// TIA Portal V17 export
// export: Created 2023-12-22T15:03:00.6243464Z, ExportSetting WithDefaults, DisplayName Totally Integrated Automation Portal, DisplayVersion V17, DisplayName TIA Portal Openness, DisplayVersion V17, DisplayName TIA Portal Version Control Interface, DisplayVersion V17, DisplayName STEP 7 Professional, DisplayVersion V17, DisplayName STEP 7 Safety, DisplayVersion V17, DisplayName WinCC Advanced, DisplayVersion V17
FUNCTION_BLOCK "DRV_M_D"   // FB110, LAD
{ S7_Optimized_Access := 'FALSE' }
VERSION : 0.1
// stored: AutoNumber false, IsIECCheckEnabled false, SetENOAutomatically false, UDAEnableTagReadback false
   VAR_INPUT
      All_Block : Bool;   // Аварийный останов
   END_VAR
   VAR_IN_OUT
      FB_QF : Bool;   // защитный автомат / Защитный автомат / Готовность
      FB_KM : Bool;   // привод запущен / Пускатель / В работе
      S_Alarm : Bool;   // Внешний индикатор наличия аварии
      CMD_Run : Bool;   // Команда запуска двигателя
   END_VAR
   VAR DB_SPECIFIC
      CMD : "CMD";   // Основные команды / Блок команд
      Mode : Int;   // Режим работы
      Status : Int;   // Статус устройства
      Use : Struct   // Функционал
         QF { S7_SetPoint := 'True'} : Bool := true;   // Защитный автомат
         KM { S7_SetPoint := 'True'} : Bool := true;   // Пускатель
         OpTime { S7_SetPoint := 'True'} : Bool := true;   // Контроль наработки
         Analog { S7_SetPoint := 'True'} : Bool;
         Local_Keys : Bool;
      END_STRUCT;
      FB : Struct   // Функционал
         QF : Bool;   // Защитный автомат
         KM : Bool;   // Пускатель
         Local_Start : Bool;
         Local_Stop : Bool;
      END_STRUCT;
      ON : Bool;   // Успешно запущено
      OFF : Bool;   // Успешно остановлено
   END_VAR
   VAR
      Tx { S7_SetPoint := 'True'} : Array[0..3] of "Time_S";   // Блок таймеров
   END_VAR
   VAR DB_SPECIFIC
      Inv : Struct   // Инверсия сигналов
         CMD { S7_SetPoint := 'True'} : Bool;   // Команда запуска
         QF { S7_SetPoint := 'True'} : Bool;   // Защитный автомат
         KM { S7_SetPoint := 'True'} : Bool;   // Пускатель
      END_STRUCT;
      Alarm : Struct   // Сбор аварий / Список аварий
         Block : Bool;   // Аварийная остановка
         QF : Bool;   // привод не готов / Выбило защитный автомат
         Start : Bool;   // Ошибка при запуске
         Stop : Bool;   // Ошибка при останове
         Termo : Bool;   // термозащита / Сработала термозащита
         Alarm : Bool;   // Внешняя авария
         Safety : Bool;   // Сработала безопасность
         OpTime : Bool;
      END_STRUCT;
      Alarms : Word;   // Слово аварий
      Events : Word;   // События
      pos : Array[0..15] of Bool;
      OpTime_h : DInt;   // наработка (ч)
      OpTime_s { S7_SetPoint := 'True'} : DInt;   // наработка (с)
      OpTime_SP { S7_SetPoint := 'True'} : DInt := 2160;   // Интервал обслуживания, ч
      OpTime_Now_h : DInt;   // Прошло с прошлого обслуживания, ч
      OpTime_Now_s { S7_SetPoint := 'True'} : DInt;   // Прошло с прошлого обслуживания, с
      CodeID { S7_SetPoint := 'True'} : Int;   // Код датчика для привязки в скаде
      Indirect : Struct   // Использование косвенной адресации
         FB_QF { S7_SetPoint := 'True'} : Bool := true;   // Защитный автомат
         FB_KM { S7_SetPoint := 'True'} : Bool := true;   // Пускатель
         CMD { S7_SetPoint := 'True'} : Bool := true;   // Запуск двигателя
      END_STRUCT;
      Indirect_BYTE : Struct   // Адрес входа на контроллере (Байт)
         FB_QF { S7_SetPoint := 'True'} : Int;   // Защитный автомат
         FB_KM { S7_SetPoint := 'True'} : Int;   // Пускатель
         CMD { S7_SetPoint := 'True'} : Int;   // Запуск двигателя
      END_STRUCT;
      Indirect_BIT : Struct   // Адрес входа на контроллере (Бит)
         FB_QF { S7_SetPoint := 'True'} : Int := 9;   // Защитный автомат
         FB_KM { S7_SetPoint := 'True'} : Int := 9;   // Пускатель
         CMD { S7_SetPoint := 'True'} : Int := 9;   // Запуск двигателя
      END_STRUCT;
      Time_DTL : DTL;
   END_VAR
   VAR_TEMP
      ev : Bool;
      xQF : Bool;
      xKM : Bool;
   END_VAR
   VAR_TEMP   // added for the SCL form of the ladder/FBD networks
      _w1 : Bool;
      _w2 : Bool;
      _w3 : Bool;
      _w4 : Bool;
      _w5 : Bool;
      _w6 : Bool;
      _w7 : Bool;
      _w8 : Bool;
      _w9 : Bool;
      _w10 : Bool;
      _w11 : Bool;
      _w12 : Bool;
      _w13 : Bool;
      _w14 : Bool;
      _w15 : Bool;
      _w16 : Bool;
      _w17 : Bool;
      _w18 : Bool;
      _w19 : Bool;
      _w20 : Bool;
      _w21 : Bool;
      _w22 : Bool;
      _w23 : Bool;
      _w24 : Bool;
      _w25 : Bool;
      _w26 : Bool;
   END_VAR
BEGIN

REGION Network 1: Режим глобальной симуляции
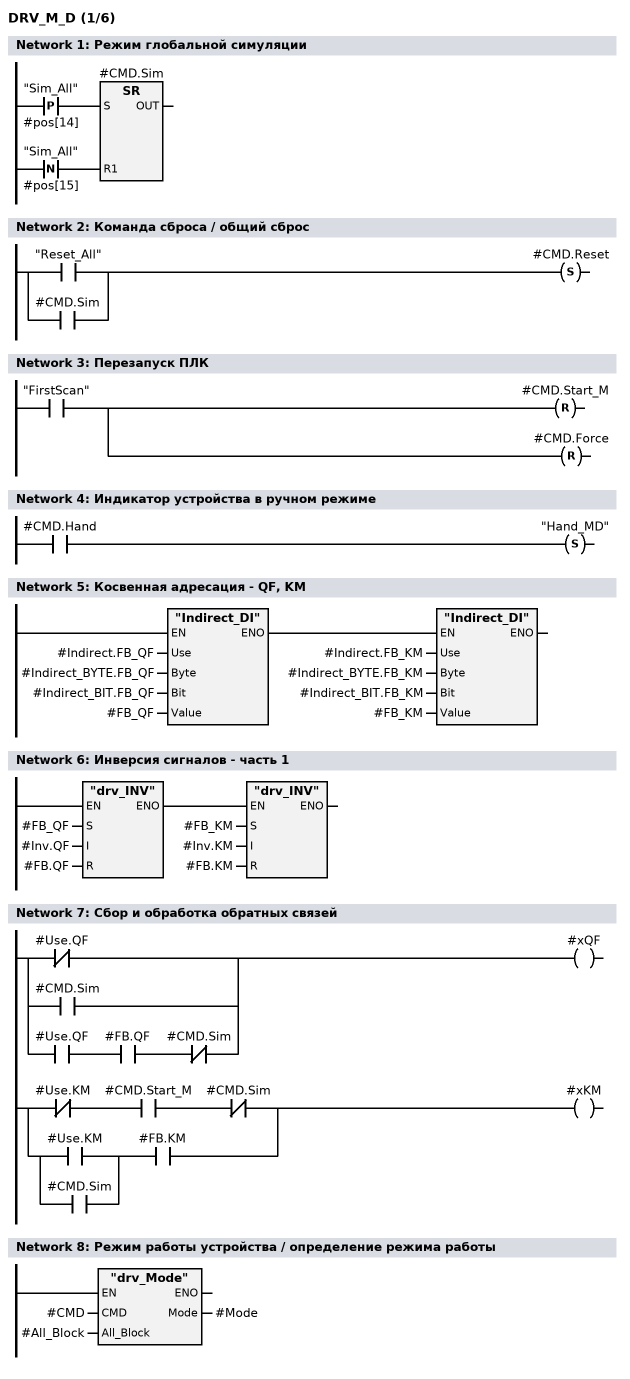
   RUNG wire#powerrail
      P_Contact(operand := "Sim_All", bit := #pos[14])
      S_SR(operand := #CMD.Sim, r1 := wire#w1)
   END_RUNG
   RUNG wire#powerrail
      N_Contact(operand := "Sim_All", bit := #pos[15])
   END_RUNG wire#w1
   // the same network as SCL:
   #_w1 := "Sim_All" AND NOT #pos[14];   // rising edge of "Sim_All"
   #pos[14] := "Sim_All";
   #_w2 := NOT "Sim_All" AND #pos[15];   // falling edge of "Sim_All"
   #pos[15] := "Sim_All";
   IF #_w1 THEN
       #CMD.Sim := TRUE;   // SR flip-flop
   END_IF;
   IF #_w2 THEN #CMD.Sim := FALSE; END_IF;
END_REGION

REGION Network 2: Команда сброса / общий сброс
   RUNG wire#powerrail
      Contact( "Reset_All" )
      wire#w1
      S_Coil( #CMD.Reset )
   END_RUNG
   RUNG wire#powerrail
      Contact( #CMD.Sim )
   END_RUNG wire#w1
   // the same network as SCL:
   IF "Reset_All" OR #CMD.Sim THEN #CMD.Reset := TRUE; END_IF;
END_REGION

REGION Network 3: Перезапуск ПЛК
   RUNG wire#powerrail
      Contact( "FirstScan" )
      wire#w1
      R_Coil( #CMD.Start_M )
   END_RUNG
   RUNG wire#w1
      R_Coil( #CMD.Force )
   END_RUNG
   // the same network as SCL:
   IF "FirstScan" THEN
       #CMD.Start_M := FALSE;
       #CMD.Force := FALSE;
   END_IF;
END_REGION

REGION Network 4: Индикатор устройства в ручном режиме
   RUNG wire#powerrail
      Contact( #CMD.Hand )
      S_Coil( "Hand_MD" )
   END_RUNG
   // the same network as SCL:
   IF #CMD.Hand THEN "Hand_MD" := TRUE; END_IF;
END_REGION

REGION Network 5: Косвенная адресация - QF, KM
   RUNG wire#powerrail
      "Indirect_DI"(Use := #Indirect.FB_QF, "Byte" := #Indirect_BYTE.FB_QF, Bit := #Indirect_BIT.FB_QF, Value := #FB_QF)
      "Indirect_DI"(Use := #Indirect.FB_KM, "Byte" := #Indirect_BYTE.FB_KM, Bit := #Indirect_BIT.FB_KM, Value := #FB_KM)
   END_RUNG
   // the same network as SCL:
   "Indirect_DI"(Use := #Indirect.FB_QF,
                 "Byte" := #Indirect_BYTE.FB_QF,
                 Bit := #Indirect_BIT.FB_QF,
                 Value := #FB_QF,
                 ENO => #_w1);
   IF #_w1 THEN
       "Indirect_DI"(Use := #Indirect.FB_KM,
                     "Byte" := #Indirect_BYTE.FB_KM,
                     Bit := #Indirect_BIT.FB_KM,
                     Value := #FB_KM);
   END_IF;
END_REGION

REGION Network 6: Инверсия сигналов - часть 1
   RUNG wire#powerrail
      "drv_INV"(S := #FB_QF, I := #Inv.QF, R := #FB.QF)
      "drv_INV"(S := #FB_KM, I := #Inv.KM, R := #FB.KM)
   END_RUNG
   // the same network as SCL:
   "drv_INV"(S := #FB_QF, I := #Inv.QF, R := #FB.QF, ENO => #_w1);
   IF #_w1 THEN "drv_INV"(S := #FB_KM, I := #Inv.KM, R := #FB.KM); END_IF;
END_REGION

REGION Network 7: Сбор и обработка обратных связей
   RUNG wire#powerrail
      I_Contact( #Use.QF )
      wire#w1
      Coil( #xQF )
   END_RUNG
   RUNG wire#powerrail
      Contact( #CMD.Sim )
   END_RUNG wire#w1
   RUNG wire#powerrail
      Contact( #Use.QF )
      Contact( #FB.QF )
      I_Contact( #CMD.Sim )
   END_RUNG wire#w1
   RUNG wire#powerrail
      I_Contact( #Use.KM )
      Contact( #CMD.Start_M )
      I_Contact( #CMD.Sim )
      wire#w2
      Coil( #xKM )
   END_RUNG
   RUNG wire#powerrail
      Contact( #Use.KM )
      wire#w3
      Contact( #FB.KM )
   END_RUNG wire#w2
   RUNG wire#powerrail
      Contact( #CMD.Sim )
   END_RUNG wire#w3
   // the same network as SCL:
   #xQF := NOT #Use.QF OR #CMD.Sim OR (#Use.QF AND #FB.QF AND NOT #CMD.Sim);
   #xKM := (NOT #Use.KM AND #CMD.Start_M AND NOT #CMD.Sim) OR ((#Use.KM OR #CMD.Sim) AND #FB.KM);
END_REGION

REGION Network 8: Режим работы устройства / определение режима работы
   RUNG wire#powerrail
      "drv_Mode"(CMD := #CMD, All_Block := #All_Block, Mode => #Mode)
   END_RUNG
   // the same network as SCL:
   "drv_Mode"(CMD := #CMD, All_Block := #All_Block, Mode => #Mode);
END_REGION

REGION Network 9: Управление запуском / дискретный управляющий сигнал
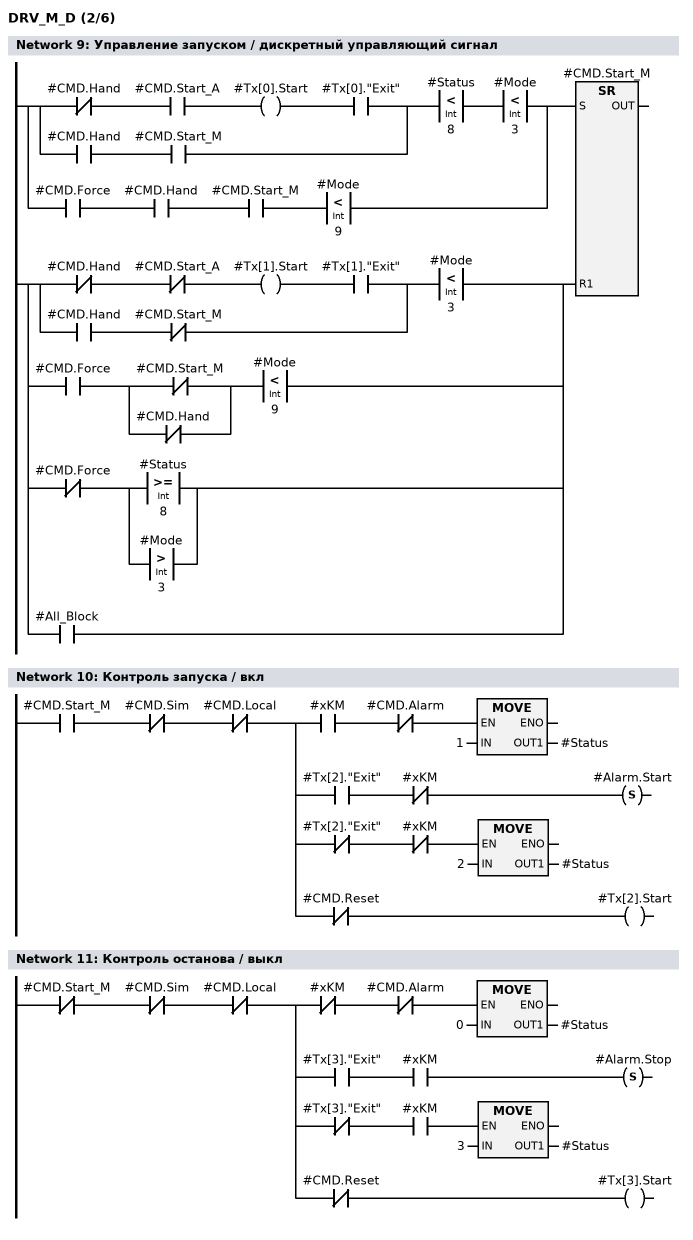
   RUNG wire#powerrail
      I_Contact( #CMD.Hand )
      Contact( #CMD.Start_A )
      Coil( #Tx[0].Start )
      Contact( #Tx[0]."Exit" )
      wire#w1
      { S7_Templates := "SrcType := Int" } LT_Contact(in1 := #Status, in2 := 8)
      { S7_Templates := "SrcType := Int" } LT_Contact(in1 := #Mode, in2 := 3)
      wire#w2
      S_SR(operand := #CMD.Start_M, r1 := wire#w7)
   END_RUNG
   RUNG wire#powerrail
      Contact( #CMD.Hand )
      Contact( #CMD.Start_M )
   END_RUNG wire#w1
   RUNG wire#powerrail
      Contact( #CMD.Force )
      Contact( #CMD.Hand )
      Contact( #CMD.Start_M )
      { S7_Templates := "SrcType := Int" } LT_Contact(in1 := #Mode, in2 := 9)
   END_RUNG wire#w2
   RUNG wire#powerrail
      I_Contact( #CMD.Hand )
      I_Contact( #CMD.Start_A )
      Coil( #Tx[1].Start )
      Contact( #Tx[1]."Exit" )
      wire#w3
      { S7_Templates := "SrcType := Int" } LT_Contact(in1 := #Mode, in2 := 3)
   END_RUNG wire#w7
   RUNG wire#powerrail
      Contact( #CMD.Hand )
      I_Contact( #CMD.Start_M )
   END_RUNG wire#w3
   RUNG wire#powerrail
      Contact( #CMD.Force )
      wire#w4
      I_Contact( #CMD.Start_M )
      wire#w5
      { S7_Templates := "SrcType := Int" } LT_Contact(in1 := #Mode, in2 := 9)
   END_RUNG wire#w7
   RUNG wire#w4
      I_Contact( #CMD.Hand )
   END_RUNG wire#w5
   RUNG wire#powerrail
      I_Contact( #CMD.Force )
      wire#w6
      { S7_Templates := "SrcType := Int" } GE_Contact(in1 := #Status, in2 := 8)
   END_RUNG wire#w7
   RUNG wire#w6
      { S7_Templates := "SrcType := Int" } GT_Contact(in1 := #Mode, in2 := 3)
   END_RUNG wire#w7
   RUNG wire#powerrail
      Contact( #All_Block )
   END_RUNG wire#w7
   // the same network as SCL:
   #Tx[0].Start := NOT #CMD.Hand AND #CMD.Start_A;
   #_w1 := (((NOT #CMD.Hand AND #CMD.Start_A AND #Tx[0]."Exit") OR (#CMD.Hand AND #CMD.Start_M)) AND (#Status < 8) AND (#Mode < 3)) OR (#CMD.Force AND #CMD.Hand AND #CMD.Start_M AND (#Mode < 9));
   #Tx[1].Start := NOT #CMD.Hand AND NOT #CMD.Start_A;
   #_w2 := (((NOT #CMD.Hand AND NOT #CMD.Start_A AND #Tx[1]."Exit") OR (#CMD.Hand AND NOT #CMD.Start_M)) AND (#Mode < 3)) OR (#CMD.Force AND (NOT #CMD.Start_M OR NOT #CMD.Hand) AND (#Mode < 9)) OR (NOT #CMD.Force AND ((#Status >= 8) OR (#Mode > 3))) OR #All_Block;
   IF #_w1 THEN
       #CMD.Start_M := TRUE;   // SR flip-flop
   END_IF;
   IF #_w2 THEN #CMD.Start_M := FALSE; END_IF;
END_REGION

REGION Network 10: Контроль запуска / вкл
   RUNG wire#powerrail
      Contact( #CMD.Start_M )
      I_Contact( #CMD.Sim )
      I_Contact( #CMD.Local )
      wire#w1
      Contact( #xKM )
      I_Contact( #CMD.Alarm )
      { S7_GenerateENO := "TRUE" } Move(in := 1, out1 => #Status)
   END_RUNG
   RUNG wire#w1
      Contact( #Tx[2]."Exit" )
      I_Contact( #xKM )
      S_Coil( #Alarm.Start )
   END_RUNG
   RUNG wire#w1
      I_Contact( #Tx[2]."Exit" )
      I_Contact( #xKM )
      { S7_GenerateENO := "TRUE" } Move(in := 2, out1 => #Status)
   END_RUNG
   RUNG wire#w1
      I_Contact( #CMD.Reset )
      Coil( #Tx[2].Start )
   END_RUNG
   // the same network as SCL:
   #_w1 := #CMD.Start_M AND NOT #CMD.Sim AND NOT #CMD.Local;
   IF #_w1 AND #xKM AND NOT #CMD.Alarm THEN #Status := 1; END_IF;
   IF #_w1 AND #Tx[2]."Exit" AND NOT #xKM THEN #Alarm.Start := TRUE; END_IF;
   IF #_w1 AND NOT #Tx[2]."Exit" AND NOT #xKM THEN #Status := 2; END_IF;
   #Tx[2].Start := #_w1 AND NOT #CMD.Reset;
END_REGION

REGION Network 11: Контроль останова / выкл
   RUNG wire#powerrail
      I_Contact( #CMD.Start_M )
      I_Contact( #CMD.Sim )
      I_Contact( #CMD.Local )
      wire#w1
      I_Contact( #xKM )
      I_Contact( #CMD.Alarm )
      { S7_GenerateENO := "TRUE" } Move(in := 0, out1 => #Status)
   END_RUNG
   RUNG wire#w1
      Contact( #Tx[3]."Exit" )
      Contact( #xKM )
      S_Coil( #Alarm.Stop )
   END_RUNG
   RUNG wire#w1
      I_Contact( #Tx[3]."Exit" )
      Contact( #xKM )
      { S7_GenerateENO := "TRUE" } Move(in := 3, out1 => #Status)
   END_RUNG
   RUNG wire#w1
      I_Contact( #CMD.Reset )
      Coil( #Tx[3].Start )
   END_RUNG
   // the same network as SCL:
   #_w1 := NOT #CMD.Start_M AND NOT #CMD.Sim AND NOT #CMD.Local;
   IF #_w1 AND NOT #xKM AND NOT #CMD.Alarm THEN #Status := 0; END_IF;
   IF #_w1 AND #Tx[3]."Exit" AND #xKM THEN #Alarm.Stop := TRUE; END_IF;
   IF #_w1 AND NOT #Tx[3]."Exit" AND #xKM THEN #Status := 3; END_IF;
   #Tx[3].Start := #_w1 AND NOT #CMD.Reset;
END_REGION

REGION Network 12: Локальный режим
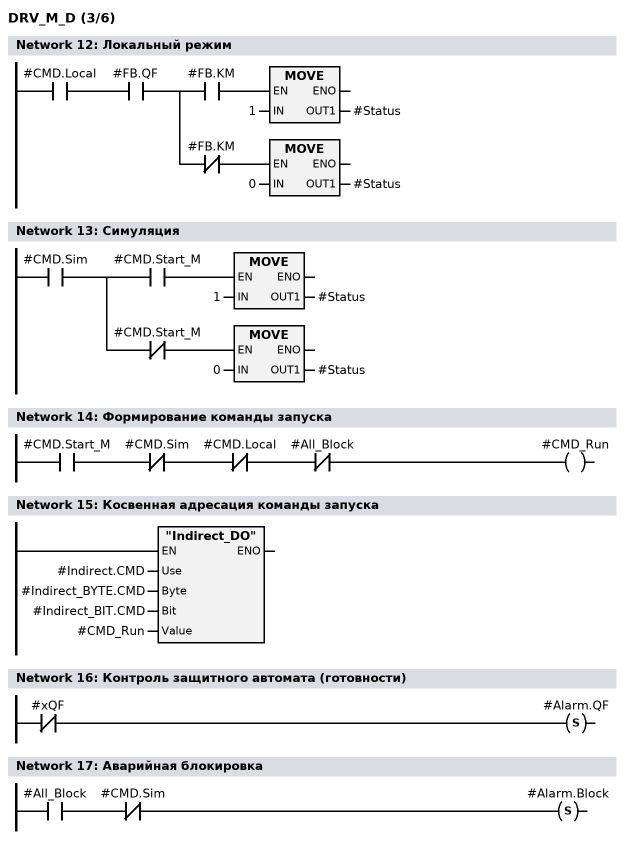
   RUNG wire#powerrail
      Contact( #CMD.Local )
      Contact( #FB.QF )
      wire#w1
      Contact( #FB.KM )
      { S7_GenerateENO := "TRUE" } Move(in := 1, out1 => #Status)
   END_RUNG
   RUNG wire#w1
      I_Contact( #FB.KM )
      { S7_GenerateENO := "TRUE" } Move(in := 0, out1 => #Status)
   END_RUNG
   // the same network as SCL:
   #_w1 := #CMD.Local AND #FB.QF;
   IF #_w1 AND #FB.KM THEN #Status := 1; END_IF;
   IF #_w1 AND NOT #FB.KM THEN #Status := 0; END_IF;
END_REGION

REGION Network 13: Симуляция
   RUNG wire#powerrail
      Contact( #CMD.Sim )
      wire#w1
      Contact( #CMD.Start_M )
      { S7_GenerateENO := "TRUE" } Move(in := 1, out1 => #Status)
   END_RUNG
   RUNG wire#w1
      I_Contact( #CMD.Start_M )
      { S7_GenerateENO := "TRUE" } Move(in := 0, out1 => #Status)
   END_RUNG
   // the same network as SCL:
   IF #CMD.Sim AND #CMD.Start_M THEN #Status := 1; END_IF;
   IF #CMD.Sim AND NOT #CMD.Start_M THEN #Status := 0; END_IF;
END_REGION

REGION Network 14: Формирование команды запуска
   RUNG wire#powerrail
      Contact( #CMD.Start_M )
      I_Contact( #CMD.Sim )
      I_Contact( #CMD.Local )
      I_Contact( #All_Block )
      Coil( #CMD_Run )
   END_RUNG
   // the same network as SCL:
   #CMD_Run := #CMD.Start_M AND NOT #CMD.Sim AND NOT #CMD.Local AND NOT #All_Block;
END_REGION

REGION Network 15: Косвенная адресация команды запуска
   RUNG wire#powerrail
      "Indirect_DO"(Use := #Indirect.CMD, "Byte" := #Indirect_BYTE.CMD, Bit := #Indirect_BIT.CMD, Value := #CMD_Run)
   END_RUNG
   // the same network as SCL:
   "Indirect_DO"(Use := #Indirect.CMD,
                 "Byte" := #Indirect_BYTE.CMD,
                 Bit := #Indirect_BIT.CMD,
                 Value := #CMD_Run);
END_REGION

REGION Network 16: Контроль защитного автомата (готовности)
   RUNG wire#powerrail
      I_Contact( #xQF )
      S_Coil( #Alarm.QF )
   END_RUNG
   // the same network as SCL:
   IF NOT #xQF THEN #Alarm.QF := TRUE; END_IF;
END_REGION

REGION Network 17: Аварийная блокировка
   RUNG wire#powerrail
      Contact( #All_Block )
      I_Contact( #CMD.Sim )
      S_Coil( #Alarm.Block )
   END_RUNG
   // the same network as SCL:
   IF #All_Block AND NOT #CMD.Sim THEN #Alarm.Block := TRUE; END_IF;
END_REGION

REGION Network 18: Сигнал аварии
   // Safety - сработал датчик безопасности, подключается через отдельный дискретный вход
   // Termo - сработала термозащита, подключается через отдельный дискретный вход
   // Alarm - сработала внешняя авария, подключается через отдельный дискретный вход
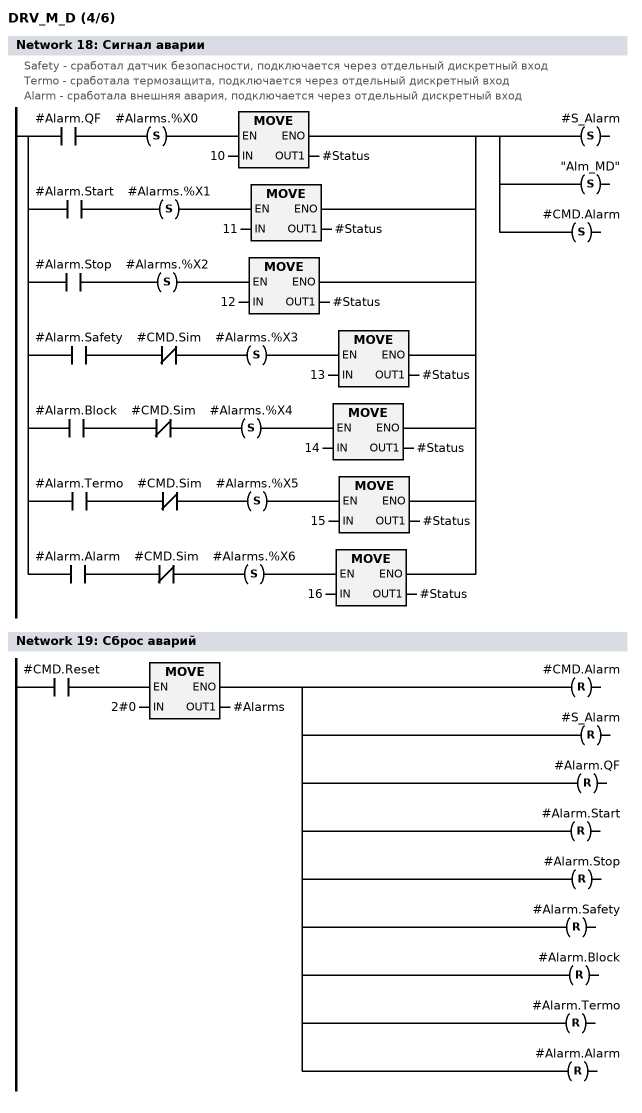
   RUNG wire#powerrail
      Contact( #Alarm.QF )
      S_Coil( #Alarms.%X0 )
      { S7_GenerateENO := "TRUE" } Move(in := 10, out1 => #Status)
      wire#w1
      S_Coil( #S_Alarm )
   END_RUNG
   RUNG wire#powerrail
      Contact( #Alarm.Start )
      S_Coil( #Alarms.%X1 )
      { S7_GenerateENO := "TRUE" } Move(in := 11, out1 => #Status)
   END_RUNG wire#w1
   RUNG wire#powerrail
      Contact( #Alarm.Stop )
      S_Coil( #Alarms.%X2 )
      { S7_GenerateENO := "TRUE" } Move(in := 12, out1 => #Status)
   END_RUNG wire#w1
   RUNG wire#powerrail
      Contact( #Alarm.Safety )
      I_Contact( #CMD.Sim )
      S_Coil( #Alarms.%X3 )
      { S7_GenerateENO := "TRUE" } Move(in := 13, out1 => #Status)
   END_RUNG wire#w1
   RUNG wire#powerrail
      Contact( #Alarm.Block )
      I_Contact( #CMD.Sim )
      S_Coil( #Alarms.%X4 )
      { S7_GenerateENO := "TRUE" } Move(in := 14, out1 => #Status)
   END_RUNG wire#w1
   RUNG wire#powerrail
      Contact( #Alarm.Termo )
      I_Contact( #CMD.Sim )
      S_Coil( #Alarms.%X5 )
      { S7_GenerateENO := "TRUE" } Move(in := 15, out1 => #Status)
   END_RUNG wire#w1
   RUNG wire#powerrail
      Contact( #Alarm.Alarm )
      I_Contact( #CMD.Sim )
      S_Coil( #Alarms.%X6 )
      { S7_GenerateENO := "TRUE" } Move(in := 16, out1 => #Status)
   END_RUNG wire#w1
   RUNG wire#w1
      S_Coil( "Alm_MD" )
   END_RUNG
   RUNG wire#w1
      S_Coil( #CMD.Alarm )
   END_RUNG
   // the same network as SCL:
   // ENO of a box is taken as its EN; it also drops when the box reports an error
   IF #Alarm.QF THEN
       #Alarms.%X0 := TRUE;
       #Status := 10;
   END_IF;
   IF #Alarm.Start THEN
       #Alarms.%X1 := TRUE;
       #Status := 11;
   END_IF;
   IF #Alarm.Stop THEN
       #Alarms.%X2 := TRUE;
       #Status := 12;
   END_IF;
   #_w1 := #Alarm.Safety AND NOT #CMD.Sim;
   IF #_w1 THEN
       #Alarms.%X3 := TRUE;
       #Status := 13;
   END_IF;
   #_w2 := #Alarm.Block AND NOT #CMD.Sim;
   IF #_w2 THEN
       #Alarms.%X4 := TRUE;
       #Status := 14;
   END_IF;
   #_w3 := #Alarm.Termo AND NOT #CMD.Sim;
   IF #_w3 THEN
       #Alarms.%X5 := TRUE;
       #Status := 15;
   END_IF;
   #_w4 := #Alarm.Alarm AND NOT #CMD.Sim;
   IF #_w4 THEN
       #Alarms.%X6 := TRUE;
       #Status := 16;
   END_IF;
   IF #Alarm.QF OR #Alarm.Start OR #Alarm.Stop OR #_w1 OR #_w2 OR #_w3 OR #_w4 THEN
       #S_Alarm := TRUE;
       "Alm_MD" := TRUE;
       #CMD.Alarm := TRUE;
   END_IF;
END_REGION

REGION Network 19: Сброс аварий
   RUNG wire#powerrail
      Contact( #CMD.Reset )
      Move(in := 2#0, out1 => #Alarms)
      wire#w1
      R_Coil( #CMD.Alarm )
   END_RUNG
   RUNG wire#w1
      R_Coil( #S_Alarm )
   END_RUNG
   RUNG wire#w1
      R_Coil( #Alarm.QF )
   END_RUNG
   RUNG wire#w1
      R_Coil( #Alarm.Start )
   END_RUNG
   RUNG wire#w1
      R_Coil( #Alarm.Stop )
   END_RUNG
   RUNG wire#w1
      R_Coil( #Alarm.Safety )
   END_RUNG
   RUNG wire#w1
      R_Coil( #Alarm.Block )
   END_RUNG
   RUNG wire#w1
      R_Coil( #Alarm.Termo )
   END_RUNG
   RUNG wire#w1
      R_Coil( #Alarm.Alarm )
   END_RUNG
   // the same network as SCL:
   IF #CMD.Reset THEN
       #Alarms := 2#0;
       #CMD.Alarm := FALSE;
       #S_Alarm := FALSE;
       #Alarm.QF := FALSE;
       #Alarm.Start := FALSE;
       #Alarm.Stop := FALSE;
       #Alarm.Safety := FALSE;
       #Alarm.Block := FALSE;
       #Alarm.Termo := FALSE;
       #Alarm.Alarm := FALSE;
   END_IF;
END_REGION

REGION Network 20: События привода
   // 0 - ручной режим активирован
   // 1 - ручной режим деактивирован
   // 2 - принудительный режим активирован
   // 3 - принудительный режим деактивирован
   // 4 - запуск в ручном режиме
   // 5 - останов в ручном режиме
   // 6 - местный режим управления активирован
   // 7 - местный режим управления деактивирован
   // 8 - запущено в местном режиме
   // 9 - остановлено в местном режиме
   // 10 - проведено сервисное обслуживание
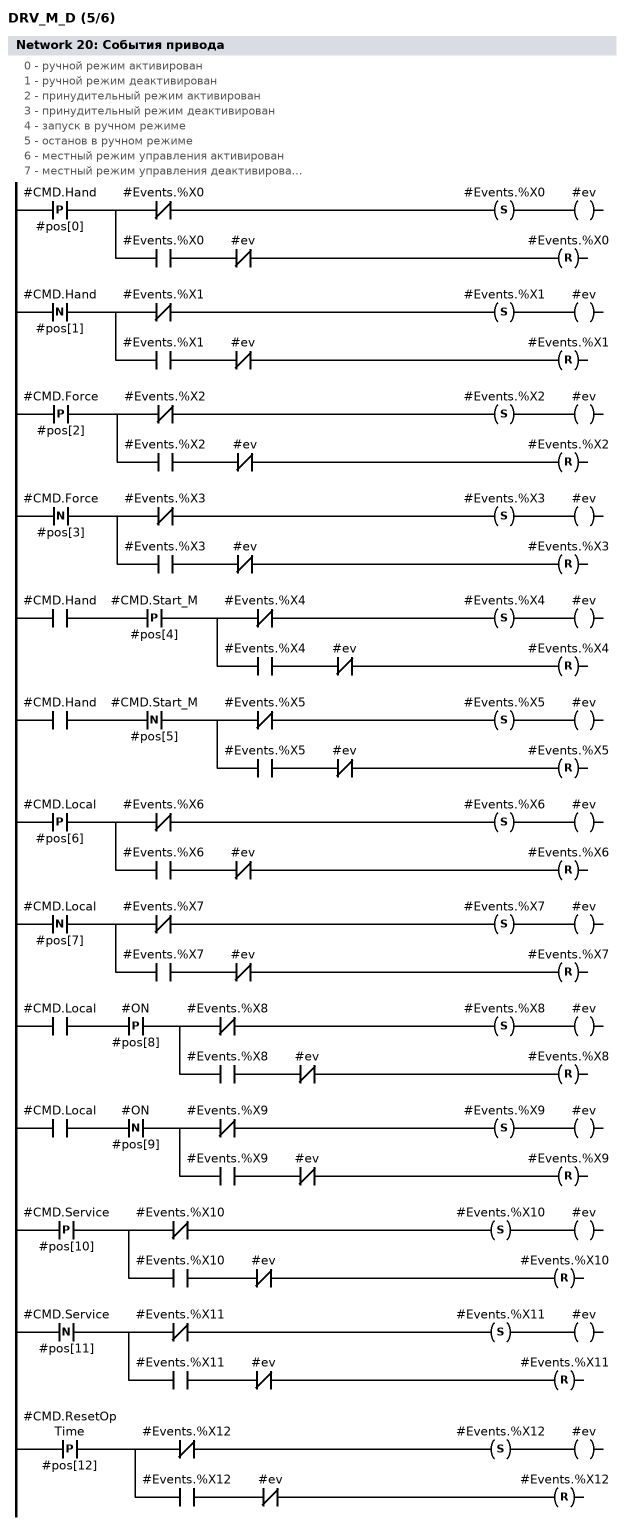
   RUNG wire#powerrail
      P_Contact(operand := #CMD.Hand, bit := #pos[0])
      wire#w1
      I_Contact( #Events.%X0 )
      S_Coil( #Events.%X0 )
      Coil( #ev )
   END_RUNG
   RUNG wire#w1
      Contact( #Events.%X0 )
      I_Contact( #ev )
      R_Coil( #Events.%X0 )
   END_RUNG
   RUNG wire#powerrail
      N_Contact(operand := #CMD.Hand, bit := #pos[1])
      wire#w2
      I_Contact( #Events.%X1 )
      S_Coil( #Events.%X1 )
      Coil( #ev )
   END_RUNG
   RUNG wire#w2
      Contact( #Events.%X1 )
      I_Contact( #ev )
      R_Coil( #Events.%X1 )
   END_RUNG
   RUNG wire#powerrail
      P_Contact(operand := #CMD.Force, bit := #pos[2])
      wire#w3
      I_Contact( #Events.%X2 )
      S_Coil( #Events.%X2 )
      Coil( #ev )
   END_RUNG
   RUNG wire#w3
      Contact( #Events.%X2 )
      I_Contact( #ev )
      R_Coil( #Events.%X2 )
   END_RUNG
   RUNG wire#powerrail
      N_Contact(operand := #CMD.Force, bit := #pos[3])
      wire#w4
      I_Contact( #Events.%X3 )
      S_Coil( #Events.%X3 )
      Coil( #ev )
   END_RUNG
   RUNG wire#w4
      Contact( #Events.%X3 )
      I_Contact( #ev )
      R_Coil( #Events.%X3 )
   END_RUNG
   RUNG wire#powerrail
      Contact( #CMD.Hand )
      P_Contact(operand := #CMD.Start_M, bit := #pos[4])
      wire#w5
      I_Contact( #Events.%X4 )
      S_Coil( #Events.%X4 )
      Coil( #ev )
   END_RUNG
   RUNG wire#w5
      Contact( #Events.%X4 )
      I_Contact( #ev )
      R_Coil( #Events.%X4 )
   END_RUNG
   RUNG wire#powerrail
      Contact( #CMD.Hand )
      N_Contact(operand := #CMD.Start_M, bit := #pos[5])
      wire#w6
      I_Contact( #Events.%X5 )
      S_Coil( #Events.%X5 )
      Coil( #ev )
   END_RUNG
   RUNG wire#w6
      Contact( #Events.%X5 )
      I_Contact( #ev )
      R_Coil( #Events.%X5 )
   END_RUNG
   RUNG wire#powerrail
      P_Contact(operand := #CMD.Local, bit := #pos[6])
      wire#w7
      I_Contact( #Events.%X6 )
      S_Coil( #Events.%X6 )
      Coil( #ev )
   END_RUNG
   RUNG wire#w7
      Contact( #Events.%X6 )
      I_Contact( #ev )
      R_Coil( #Events.%X6 )
   END_RUNG
   RUNG wire#powerrail
      N_Contact(operand := #CMD.Local, bit := #pos[7])
      wire#w8
      I_Contact( #Events.%X7 )
      S_Coil( #Events.%X7 )
      Coil( #ev )
   END_RUNG
   RUNG wire#w8
      Contact( #Events.%X7 )
      I_Contact( #ev )
      R_Coil( #Events.%X7 )
   END_RUNG
   RUNG wire#powerrail
      Contact( #CMD.Local )
      P_Contact(operand := #ON, bit := #pos[8])
      wire#w9
      I_Contact( #Events.%X8 )
      S_Coil( #Events.%X8 )
      Coil( #ev )
   END_RUNG
   RUNG wire#w9
      Contact( #Events.%X8 )
      I_Contact( #ev )
      R_Coil( #Events.%X8 )
   END_RUNG
   RUNG wire#powerrail
      Contact( #CMD.Local )
      N_Contact(operand := #ON, bit := #pos[9])
      wire#w10
      I_Contact( #Events.%X9 )
      S_Coil( #Events.%X9 )
      Coil( #ev )
   END_RUNG
   RUNG wire#w10
      Contact( #Events.%X9 )
      I_Contact( #ev )
      R_Coil( #Events.%X9 )
   END_RUNG
   RUNG wire#powerrail
      P_Contact(operand := #CMD.Service, bit := #pos[10])
      wire#w11
      I_Contact( #Events.%X10 )
      S_Coil( #Events.%X10 )
      Coil( #ev )
   END_RUNG
   RUNG wire#w11
      Contact( #Events.%X10 )
      I_Contact( #ev )
      R_Coil( #Events.%X10 )
   END_RUNG
   RUNG wire#powerrail
      N_Contact(operand := #CMD.Service, bit := #pos[11])
      wire#w12
      I_Contact( #Events.%X11 )
      S_Coil( #Events.%X11 )
      Coil( #ev )
   END_RUNG
   RUNG wire#w12
      Contact( #Events.%X11 )
      I_Contact( #ev )
      R_Coil( #Events.%X11 )
   END_RUNG
   RUNG wire#powerrail
      P_Contact(operand := #CMD.ResetOpTime, bit := #pos[12])
      wire#w13
      I_Contact( #Events.%X12 )
      S_Coil( #Events.%X12 )
      Coil( #ev )
   END_RUNG
   RUNG wire#w13
      Contact( #Events.%X12 )
      I_Contact( #ev )
      R_Coil( #Events.%X12 )
   END_RUNG
   // the same network as SCL:
   #_w1 := #CMD.Hand AND NOT #pos[0];   // rising edge of #CMD.Hand
   #pos[0] := #CMD.Hand;
   #_w2 := #_w1 AND NOT #Events.%X0;
   IF #_w2 THEN #Events.%X0 := TRUE; END_IF;
   #ev := #_w2;
   IF #_w1 AND #Events.%X0 AND NOT #ev THEN #Events.%X0 := FALSE; END_IF;
   #_w3 := NOT #CMD.Hand AND #pos[1];   // falling edge of #CMD.Hand
   #pos[1] := #CMD.Hand;
   #_w4 := #_w3 AND NOT #Events.%X1;
   IF #_w4 THEN #Events.%X1 := TRUE; END_IF;
   #ev := #_w4;
   IF #_w3 AND #Events.%X1 AND NOT #ev THEN #Events.%X1 := FALSE; END_IF;
   #_w5 := #CMD.Force AND NOT #pos[2];   // rising edge of #CMD.Force
   #pos[2] := #CMD.Force;
   #_w6 := #_w5 AND NOT #Events.%X2;
   IF #_w6 THEN #Events.%X2 := TRUE; END_IF;
   #ev := #_w6;
   IF #_w5 AND #Events.%X2 AND NOT #ev THEN #Events.%X2 := FALSE; END_IF;
   #_w7 := NOT #CMD.Force AND #pos[3];   // falling edge of #CMD.Force
   #pos[3] := #CMD.Force;
   #_w8 := #_w7 AND NOT #Events.%X3;
   IF #_w8 THEN #Events.%X3 := TRUE; END_IF;
   #ev := #_w8;
   IF #_w7 AND #Events.%X3 AND NOT #ev THEN #Events.%X3 := FALSE; END_IF;
   #_w9 := #CMD.Hand AND #CMD.Start_M AND NOT #pos[4];   // rising edge of #CMD.Start_M
   #pos[4] := #CMD.Start_M;
   #_w10 := #_w9 AND NOT #Events.%X4;
   IF #_w10 THEN #Events.%X4 := TRUE; END_IF;
   #ev := #_w10;
   IF #_w9 AND #Events.%X4 AND NOT #ev THEN #Events.%X4 := FALSE; END_IF;
   #_w11 := #CMD.Hand AND NOT #CMD.Start_M AND #pos[5];   // falling edge of #CMD.Start_M
   #pos[5] := #CMD.Start_M;
   #_w12 := #_w11 AND NOT #Events.%X5;
   IF #_w12 THEN #Events.%X5 := TRUE; END_IF;
   #ev := #_w12;
   IF #_w11 AND #Events.%X5 AND NOT #ev THEN #Events.%X5 := FALSE; END_IF;
   #_w13 := #CMD.Local AND NOT #pos[6];   // rising edge of #CMD.Local
   #pos[6] := #CMD.Local;
   #_w14 := #_w13 AND NOT #Events.%X6;
   IF #_w14 THEN #Events.%X6 := TRUE; END_IF;
   #ev := #_w14;
   IF #_w13 AND #Events.%X6 AND NOT #ev THEN #Events.%X6 := FALSE; END_IF;
   #_w15 := NOT #CMD.Local AND #pos[7];   // falling edge of #CMD.Local
   #pos[7] := #CMD.Local;
   #_w16 := #_w15 AND NOT #Events.%X7;
   IF #_w16 THEN #Events.%X7 := TRUE; END_IF;
   #ev := #_w16;
   IF #_w15 AND #Events.%X7 AND NOT #ev THEN #Events.%X7 := FALSE; END_IF;
   #_w17 := #CMD.Local AND #ON AND NOT #pos[8];   // rising edge of #ON
   #pos[8] := #ON;
   #_w18 := #_w17 AND NOT #Events.%X8;
   IF #_w18 THEN #Events.%X8 := TRUE; END_IF;
   #ev := #_w18;
   IF #_w17 AND #Events.%X8 AND NOT #ev THEN #Events.%X8 := FALSE; END_IF;
   #_w19 := #CMD.Local AND NOT #ON AND #pos[9];   // falling edge of #ON
   #pos[9] := #ON;
   #_w20 := #_w19 AND NOT #Events.%X9;
   IF #_w20 THEN #Events.%X9 := TRUE; END_IF;
   #ev := #_w20;
   IF #_w19 AND #Events.%X9 AND NOT #ev THEN #Events.%X9 := FALSE; END_IF;
   #_w21 := #CMD.Service AND NOT #pos[10];   // rising edge of #CMD.Service
   #pos[10] := #CMD.Service;
   #_w22 := #_w21 AND NOT #Events.%X10;
   IF #_w22 THEN #Events.%X10 := TRUE; END_IF;
   #ev := #_w22;
   IF #_w21 AND #Events.%X10 AND NOT #ev THEN #Events.%X10 := FALSE; END_IF;
   #_w23 := NOT #CMD.Service AND #pos[11];   // falling edge of #CMD.Service
   #pos[11] := #CMD.Service;
   #_w24 := #_w23 AND NOT #Events.%X11;
   IF #_w24 THEN #Events.%X11 := TRUE; END_IF;
   #ev := #_w24;
   IF #_w23 AND #Events.%X11 AND NOT #ev THEN #Events.%X11 := FALSE; END_IF;
   #_w25 := #CMD.ResetOpTime AND NOT #pos[12];   // rising edge of #CMD.ResetOpTime
   #pos[12] := #CMD.ResetOpTime;
   #_w26 := #_w25 AND NOT #Events.%X12;
   IF #_w26 THEN #Events.%X12 := TRUE; END_IF;
   #ev := #_w26;
   IF #_w25 AND #Events.%X12 AND NOT #ev THEN #Events.%X12 := FALSE; END_IF;
END_REGION

REGION Network 21: Сервисный режим
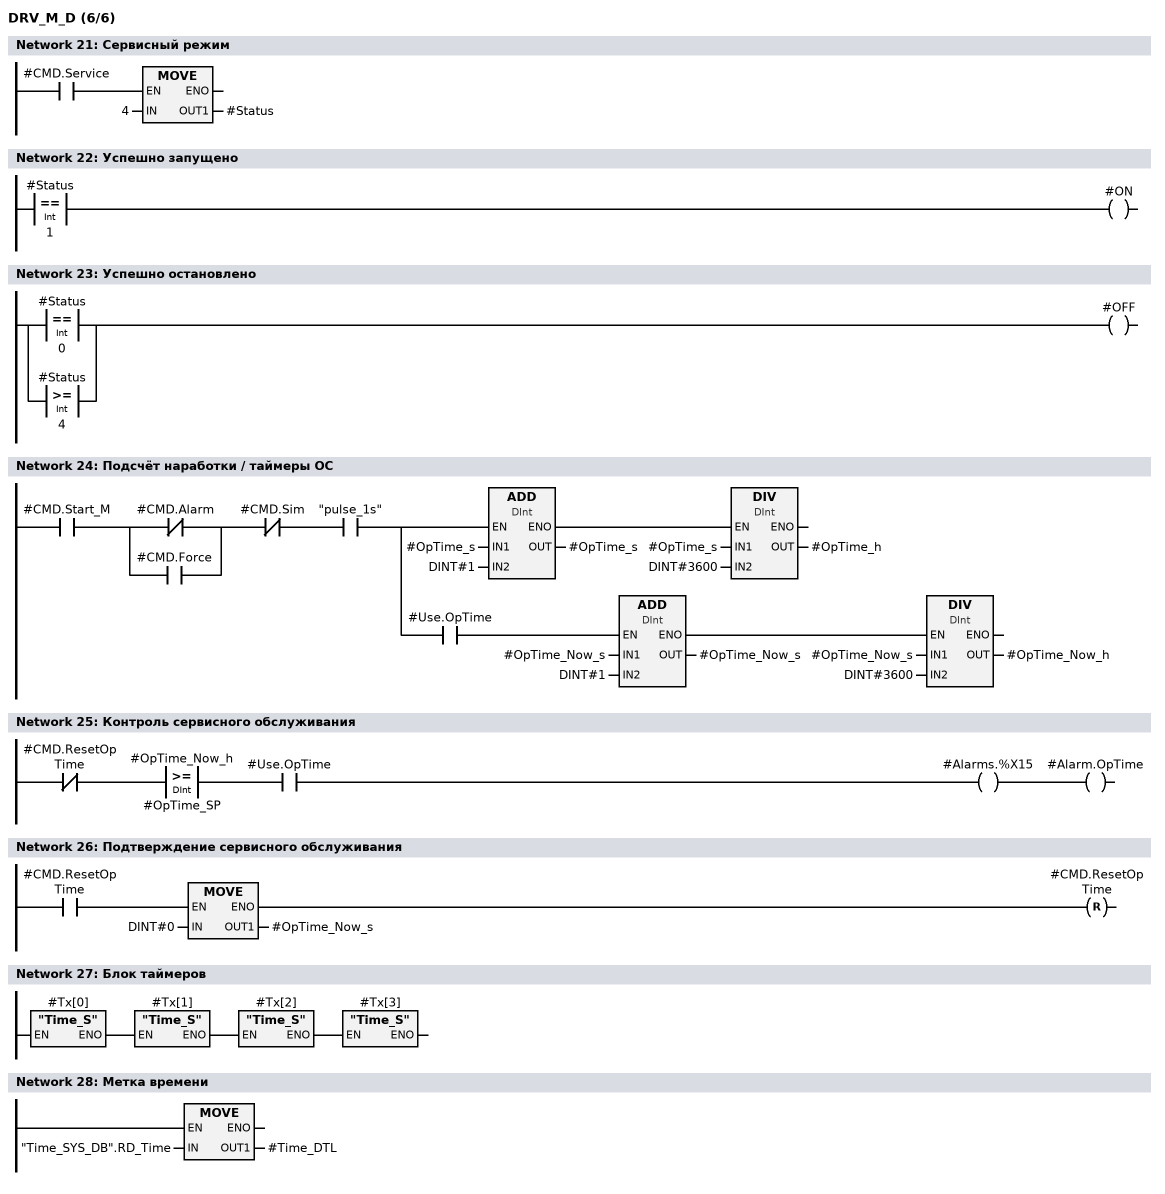
   RUNG wire#powerrail
      Contact( #CMD.Service )
      { S7_GenerateENO := "TRUE" } Move(in := 4, out1 => #Status)
   END_RUNG
   // the same network as SCL:
   IF #CMD.Service THEN #Status := 4; END_IF;
END_REGION

REGION Network 22: Успешно запущено
   RUNG wire#powerrail
      { S7_Templates := "SrcType := Int" } EQ_Contact(in1 := #Status, in2 := 1)
      Coil( #ON )
   END_RUNG
   // the same network as SCL:
   #ON := #Status = 1;
END_REGION

REGION Network 23: Успешно остановлено
   RUNG wire#powerrail
      { S7_Templates := "SrcType := Int" } EQ_Contact(in1 := #Status, in2 := 0)
      wire#w1
      Coil( #OFF )
   END_RUNG
   RUNG wire#powerrail
      { S7_Templates := "SrcType := Int" } GE_Contact(in1 := #Status, in2 := 4)
   END_RUNG wire#w1
   // the same network as SCL:
   #OFF := (#Status = 0) OR (#Status >= 4);
END_REGION

REGION Network 24: Подсчёт наработки / таймеры ОС
   RUNG wire#powerrail
      Contact( #CMD.Start_M )
      wire#w1
      I_Contact( #CMD.Alarm )
      wire#w2
      I_Contact( #CMD.Sim )
      Contact( "pulse_1s" )
      wire#w3
      { S7_Templates := "SrcType := DInt"; S7_GenerateENO := "TRUE" } Add(in1 := #OpTime_s, in2 := DINT#1, out => #OpTime_s)
      { S7_Templates := "SrcType := DInt"; S7_GenerateENO := "TRUE" } Div(in1 := #OpTime_s, in2 := DINT#3600, out => #OpTime_h)
   END_RUNG
   RUNG wire#w1
      Contact( #CMD.Force )
   END_RUNG wire#w2
   RUNG wire#w3
      Contact( #Use.OpTime )
      { S7_Templates := "SrcType := DInt"; S7_GenerateENO := "TRUE" } Add(in1 := #OpTime_Now_s, in2 := DINT#1, out => #OpTime_Now_s)
      { S7_Templates := "SrcType := DInt"; S7_GenerateENO := "TRUE" } Div(in1 := #OpTime_Now_s, in2 := DINT#3600, out => #OpTime_Now_h)
   END_RUNG
   // the same network as SCL:
   // ENO of a box is taken as its EN; it also drops when the box reports an error
   #_w1 := #CMD.Start_M AND (NOT #CMD.Alarm OR #CMD.Force) AND NOT #CMD.Sim AND "pulse_1s";
   IF #_w1 THEN
       #OpTime_s := #OpTime_s + DINT#1;
       #OpTime_h := #OpTime_s / DINT#3600;
   END_IF;
   IF #_w1 AND #Use.OpTime THEN
       #OpTime_Now_s := #OpTime_Now_s + DINT#1;
       #OpTime_Now_h := #OpTime_Now_s / DINT#3600;
   END_IF;
END_REGION

REGION Network 25: Контроль сервисного обслуживания
   RUNG wire#powerrail
      I_Contact( #CMD.ResetOpTime )
      { S7_Templates := "SrcType := DInt" } GE_Contact(in1 := #OpTime_Now_h, in2 := #OpTime_SP)
      Contact( #Use.OpTime )
      Coil( #Alarms.%X15 )
      Coil( #Alarm.OpTime )
   END_RUNG
   // the same network as SCL:
   #Alarms.%X15 := NOT #CMD.ResetOpTime AND (#OpTime_Now_h >= #OpTime_SP) AND #Use.OpTime;
   #Alarm.OpTime := #Alarms.%X15;
END_REGION

REGION Network 26: Подтверждение сервисного обслуживания
   RUNG wire#powerrail
      Contact( #CMD.ResetOpTime )
      { S7_GenerateENO := "TRUE" } Move(in := DINT#0, out1 => #OpTime_Now_s)
      R_Coil( #CMD.ResetOpTime )
   END_RUNG
   // the same network as SCL:
   // ENO of a box is taken as its EN; it also drops when the box reports an error
   IF #CMD.ResetOpTime THEN
       #OpTime_Now_s := DINT#0;
       #CMD.ResetOpTime := FALSE;
   END_IF;
END_REGION

REGION Network 27: Блок таймеров
   RUNG wire#powerrail
      #Tx[0]()
      #Tx[1]()
      #Tx[2]()
      #Tx[3]()
   END_RUNG
   // the same network as SCL:
   #Tx[0](ENO => #_w1);   // "Time_S"
   #Tx[1](EN := #_w1, ENO => #_w2);   // "Time_S"
   #Tx[2](EN := #_w2, ENO => #_w3);   // "Time_S"
   IF #_w3 THEN
       #Tx[3]();   // "Time_S"
   END_IF;
END_REGION

REGION Network 28: Метка времени
   RUNG wire#powerrail
      Move(in := "Time_SYS_DB".RD_Time, out1 => #Time_DTL)
   END_RUNG
   // the same network as SCL:
   #Time_DTL := "Time_SYS_DB".RD_Time;
END_REGION
END_FUNCTION_BLOCK
